// TIA Portal V16 program export: 2 tag tables, 0 data types, 0 data blocks, 2 code blocks (in call order from the OBs), 4 instance data blocks

VAR_GLOBAL   // PLC tag table "Standard-Variablentabelle"
   Clock_Byte AT %MB0 : Byte;
   Clock_10Hz AT %M0.0 : Bool;
   Clock_5Hz AT %M0.1 : Bool;
   "Clock_2.5Hz" AT %M0.2 : Bool;
   Clock_2Hz AT %M0.3 : Bool;
   "Clock_1.25Hz" AT %M0.4 : Bool;
   Clock_1Hz AT %M0.5 : Bool;
   "Clock_0.625Hz" AT %M0.6 : Bool;
   "Clock_0.5Hz" AT %M0.7 : Bool;
   Status AT %MW2 : Int;
   Awaria_Potwierdzona AT %M1.0 : Bool;
   System_Pracuje AT %M1.1 : Bool;
   Reset_Potwierdzony AT %M1.2 : Bool;
   Awaria_Aktywna AT %M1.3 : Bool;
   state AT %MW4 : Int;
   Pamiec_Typ_4 AT %M1.4 : Bool;
   Pamiec_Typ_1 AT %M1.5 : Bool;
END_VAR

VAR_GLOBAL   // PLC tag table "Tag table from XML_1"
   "Sensor 1" AT %I0.0 : Bool;
   "Pusher 1 front" AT %I0.1 : Bool;
   "Pusher 1 back" AT %I0.2 : Bool;
   "At pusher 1 exit" AT %I0.3 : Bool;
   "Sensor 2" AT %I0.4 : Bool;
   "Pusher 2 front" AT %I0.5 : Bool;
   "Pusher 2 back" AT %I0.6 : Bool;
   "At pusher 2 exit" AT %I0.7 : Bool;
   Start AT %I1.0 : Bool;
   Reset AT %I1.1 : Bool;
   Stop AT %I1.2 : Bool;
   "Emergency stop" AT %I1.3 : Bool;
   "FACTORY I/O (Uruchomiony)" AT %I1.4 : Bool;
   "Entry conveyor 1" AT %Q0.0 : Bool;
   "Pusher 1" AT %Q0.1 : Bool;
   "Conveyor 1" AT %Q0.2 : Bool;
   "Entry conveyor 2" AT %Q0.3 : Bool;
   "Pusher 2" AT %Q0.4 : Bool;
   "Conveyor 2" AT %Q0.5 : Bool;
   "Start light" AT %Q0.6 : Bool;
   "Reset light" AT %Q0.7 : Bool;
   "Stop light" AT %Q1.0 : Bool;
   "Vision sensor 1" AT %ID30 : DInt;
   "Vision sensor 2" AT %ID34 : DInt;
   "Counter 1" AT %QD30 : DInt;
   "Counter 2" AT %QD34 : DInt;
END_VAR

ORGANIZATION_BLOCK "Main"   // OB1, LAD, ProgramCycle
TITLE = "Main Program Sweep (Cycle)"
{ S7_Optimized_Access := 'TRUE' }
VERSION : 0.1
// stored: AutoNumber true, IsIECCheckEnabled false, SetENOAutomatically false
   VAR_INPUT
      Initial_Call : Bool;   // Initial call of this OB
      Remanence : Bool;   // =True, if remanent data are available
   END_VAR
   VAR_TEMP
      temp : Real;
   END_VAR
BEGIN

REGION Network 1
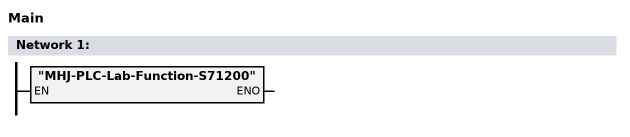
   RUNG wire#powerrail
      "MHJ-PLC-Lab-Function-S71200"()
   END_RUNG
   // the same network as SCL:
   "MHJ-PLC-Lab-Function-S71200"();
END_REGION
END_ORGANIZATION_BLOCK

ORGANIZATION_BLOCK "SCL"
TITLE = "Main Program Sweep (Cycle)"
{ S7_Optimized_Access := 'TRUE' }
VERSION : 0.1
   VAR_TEMP 
      Temp_1 : Bool;
   END_VAR


BEGIN
	// 1. LOGIKA PAMIĘCI AWARII (LATCH)
	// Jeśli wciśnięto E-Stop, ustawiamy stan awarii. 
	// Stan ten trwa nawet po wyciśnięciu E-Stop, aż do naciśnięcia Reset.
	IF NOT "Emergency stop" THEN
	    "Awaria_Aktywna" := 1;
	END_IF;
	
	IF "Reset" AND "Emergency stop" THEN
	    "Awaria_Aktywna" := 0; // Kasowanie awarii tylko gdy grzybek jest wyciśnięty
	END_IF;
	
	// 2. LOGIKA PRACY (START/STOP)
	// System może pracować tylko gdy nie ma aktywnej awarii
	IF "Start" AND NOT "Awaria_Aktywna" AND "Stop" AND "Emergency stop" THEN
	    "System_Pracuje" := 1;
	ELSIF NOT "Stop" OR "Awaria_Aktywna" THEN
	    "System_Pracuje" := 0;
	END_IF;
	
	// 3. STEROWANIE LAMPKAMI
	
	// --- LAMPKA RESET ---
	IF "Awaria_Aktywna" THEN
	    "Reset light" := "Clock_1Hz"; // Miga dopóki nie wciśniesz Reset
	ELSE
	    "Reset light" := 0;
	END_IF;
	
	// --- LAMPKA START (ZIELONA) ---
	IF "System_Pracuje" THEN
	    "Start light" := 1;           // Pali się ciągle podczas pracy
	ELSIF NOT "Awaria_Aktywna" AND "Emergency stop" AND "Stop" THEN
	    "Start light" := "Clock_1Hz"; // Miga po Resecie (gotowość do Startu)
	ELSE
	    "Start light" := 0;           // Ciemna podczas awarii
	END_IF;
	
	// --- LAMPKA STOP (CZERWONA) ---
	IF NOT "System_Pracuje" THEN
	    "Stop light" := 1;
	ELSE
	    "Stop light" := 0;
	END_IF;
	
	
	
	// 1. DETEKCJA ZBOCZY
	"F_TRIG_sensor1"(CLK := "Sensor 1");         // Zjazd z sensora zatrzymania T1
	"F_TRIG_sensor2"(CLK := "Sensor 2");         // Zjazd z sensora zatrzymania T2
	
	// Zmiana na F_TRIG dla czujników wyjściowych (zliczanie po przejechaniu elementu)
	"F_TRIG_puscher1"(CLK:="At pusher 1 exit");
	"F_TRIG_puscher2"(CLK:="At pusher 2 exit");
	
	
	// 2. OBSŁUGA LICZNIKÓW (Zliczanie na zboczu opadającym)
	IF "F_TRIG_puscher1".Q THEN
	    "Counter 1" := "Counter 1" + 1; // Element 4 został poprawnie odrzucony
	END_IF;
	
	IF "F_TRIG_puscher2".Q THEN
	    "Counter 2":= "Counter 2" + 1; // Element 1 został poprawnie odrzucony
	END_IF;
	
	// Wspólny reset liczników
	IF "Reset" THEN
	    "Counter 1" := 0;
	    "Counter 2" := 0;
	END_IF;
	
	
	
	// 3. Rejestracja typów z wizji
	IF "Vision sensor 1" = 4 THEN
	    "Pamiec_Typ_4" := 1;
	END_IF;
	IF "Vision sensor 2" = 1 THEN
	    "Pamiec_Typ_1" := 1;
	END_IF;
	
	// 4. Logika pracy sekwencyjnej
	IF "System_Pracuje" THEN
	    CASE "state" OF
	            
	        0: // --- ETAP 1: PRACA TASMY 1 (Czekanie na 4) ---
	            "Entry conveyor 1" := 1;
	            "Conveyor 1" := 1;
	            "Entry conveyor 2" := 0;
	            "Conveyor 2" := 0; // Tasma 2 stoi i czeka
	            "Pusher 1" := 0;
	            "Pusher 2" := 0;
	            
	            // Jeśli wykryto czwórkę na sensorze 1
	            IF "Pamiec_Typ_4" AND "F_TRIG_sensor1".Q THEN
	                "Entry conveyor 1" := 0;
	                "Conveyor 1" := 0;
	                "state" := 10;
	            END_IF;
	            
	        10: // --- WYPYCHANIE 4 (Z T1 na T2) ---
	            "Pusher 1" := 1;
	            IF "Pusher 1 front" THEN
	                "state" := 11;
	            END_IF;
	            
	        11: // Powrót Pushera 1 i zmiana zmiany
	            "Pusher 1" := 0;
	            IF "Pusher 1 back" THEN
	                "Pamiec_Typ_4" := 0;
	                "state" := 20; // PRZEKAZANIE PRACY DO TASMY 2
	            END_IF;
	            
	        20: // --- ETAP 2: PRACA TASMY 2 (Czekanie na 1) ---
	            "Entry conveyor 1" := 0;
	            "Conveyor 1" := 0; // Tasma 1 teraz stoi i czeka
	            "Entry conveyor 2" := 1;
	            "Conveyor 2" := 1; // Tasma 2 rusza
	            
	            // Jeśli wykryto jedynkę na sensorze 2
	            IF "Pamiec_Typ_1" AND "F_TRIG_sensor2".Q THEN
	                "Entry conveyor 2" := 0;
	                "Conveyor 2" := 0;
	                "state" := 30;
	            END_IF;
	            
	        30: // --- WYPYCHANIE 1 (Z T2 na T1) ---
	            "Pusher 2" := 1;
	            IF "Pusher 2 front" THEN
	                "state" := 31;
	            END_IF;
	            
	        31: // Powrót Pushera 2 i powrót do początku
	            "Pusher 2" := 0;
	            IF "Pusher 2 back" THEN
	                "Pamiec_Typ_1" := 0;
	                "state" := 0; // POWRÓT DO TASMY 1
	            END_IF;
	            
	    END_CASE;
	ELSE
	    // STOP
	    "Entry conveyor 1" := 0;
	    "Conveyor 1" := 0;
	    "Entry conveyor 2" := 0;
	    "Conveyor 2" := 0;
	    "Pusher 1" := 0;
	    "Pusher 2" := 0;
	    "state" := 0;
	END_IF;
	
END_ORGANIZATION_BLOCK

DATA_BLOCK "F_TRIG_puscher1"   // DB3
// stored: AutoNumber true, InstanceOfName F_TRIG, OfSystemLibElement F_TRIG, OfSystemLibVersion 1.0
"F_TRIG"
   // VAR_INPUT
   //    CLK : Bool;
   // END_VAR
   // VAR_OUTPUT
   //    Q : Bool;
   // END_VAR
   // VAR
   //    Stat_Bit : Bool;
   // END_VAR
BEGIN
END_DATA_BLOCK

DATA_BLOCK "F_TRIG_puscher2"   // DB4
// stored: AutoNumber true, InstanceOfName F_TRIG, OfSystemLibElement F_TRIG, OfSystemLibVersion 1.0
"F_TRIG"
   // VAR_INPUT
   //    CLK : Bool;
   // END_VAR
   // VAR_OUTPUT
   //    Q : Bool;
   // END_VAR
   // VAR
   //    Stat_Bit : Bool;
   // END_VAR
BEGIN
END_DATA_BLOCK

DATA_BLOCK "F_TRIG_sensor1"   // DB1
// stored: AutoNumber true, InstanceOfName F_TRIG, OfSystemLibElement F_TRIG, OfSystemLibVersion 1.0
"F_TRIG"
   // VAR_INPUT
   //    CLK : Bool;
   // END_VAR
   // VAR_OUTPUT
   //    Q : Bool;
   // END_VAR
   // VAR
   //    Stat_Bit : Bool;
   // END_VAR
BEGIN
END_DATA_BLOCK

DATA_BLOCK "F_TRIG_sensor2"   // DB2
// stored: AutoNumber true, InstanceOfName F_TRIG, OfSystemLibElement F_TRIG, OfSystemLibVersion 1.0
"F_TRIG"
   // VAR_INPUT
   //    CLK : Bool;
   // END_VAR
   // VAR_OUTPUT
   //    Q : Bool;
   // END_VAR
   // VAR
   //    Stat_Bit : Bool;
   // END_VAR
BEGIN
END_DATA_BLOCK
